FUNCTION_BLOCK FB_ALPHA215C_Multiplex EXTENDS FB_Alpha215C
(*This FB Add Messages to sign and cycle though multiple messages. Idealy One FB per Sign. 
Otherwise some messages will display longer in some signs.

st_message
- message 	(string)
- duration	(time)

*)
VAR_INPUT
END_VAR
VAR_IN_OUT
	aMessages : ARRAY [*] OF E_ALPHA_MULTIPLEX_ITEM;
END_VAR
VAR
	iCurrentItem : DINT :=  LOWER_BOUND(aMessages,1);
	iMultiplexState : UINT := 10;
	tTimer : TON;
	stItem : E_ALPHA_MULTIPLEX_ITEM;
	
END_VAR

SUPER^();

tTimer(IN:=TRUE);

CASE iMultiplexState OF
	10: // START PRINTING
		stItem := aMessages[iCurrentItem];
		
		IF stItem.bActive THEN
			SUPER^.M_Print(sAddress := stItem.sAddress,
				iFile := stItem.sFile, 
				sMessage := stItem.sMessage
			);
	
			tTimer.PT := stItem.tTime;
		ELSE
			tTimer.PT := T#0S;
		END_IF
		
		tTimer.IN := FALSE; // START TIMER
		tTimer();
		iMultiplexState := 20;
		
	20: // Wait
		IF tTimer.Q THEN //
			iCurrentItem := iCurrentItem + 1;
			
			IF iCurrentItem > UPPER_BOUND(aMessages, 1) THEN
				iCurrentItem := LOWER_BOUND(aMessages,1);
			END_IF
			iMultiplexState := 10;
		END_IF
	
END_CASE

END_FUNCTION_BLOCK

(* stored: Version 1.1.0.1
   POU FB_ALPHA215C_Multiplex: Id {0f0eb6b3-e274-4be2-b734-0d5f207bdfb1}, SpecialFunc None *)
